TYPE Newton : LREAL;
END_TYPE

(* stored: Version 1.1.0.1, ProductVersion 3.1.4024.12
   DUT Newton: Id {311c2f99-3e8f-47be-87db-aff29cae464b} *)
